{attribute addProperty BoxType "KL3102"}
{attribute addProperty Id "Channel_1Channel_B0A8062F00Channel_2Channel_B0A8062F00"}
{attribute addProperty CRC "3175726068"}
{attribute addProperty SizeInBites "0"}
{attribute addProperty SizeInBytes "0"}
TYPE KL3102_BD49BBF4 :
STRUCT
	{attribute addProperty Name "Channel_1"}
	Channel_1 : Channel_B0A8062F;
	{attribute addProperty Name "Channel_2"}
	Channel_2 : Channel_B0A8062F;
END_STRUCT
END_TYPE

(* stored: Version 1.2.0.0, ProductVersion 3.1.4024.9
   DUT KL3102_BD49BBF4: Id {fc31efd5-b727-4b31-b1ed-9b7741912cfb} *)
